TYPE ANA_Standard :
STRUCT
	MesData : ANA; (* Child structure*)

END_STRUCT
END_TYPE

(* stored: Version 1.1.0.1, ProductVersion 3.1.4024.11
   DUT ANA_Standard: Id {2d4e4e3a-4af5-4ceb-9915-b8c822facc67} *)
